PROGRAM FB_ApagadoCintas
VAR
END_VAR

IF POU_Contadores.iCintaProcesando = 0 THEN
	GVL_General.sBeltConveyor.bCintaAzul1 	:= FALSE;
	GVL_General.sBeltConveyor.bCintaVerde1	:= FALSE;
	GVL_General.sBeltConveyor.bCintaMetal1 	:= FALSE;
	GVL_General.sBeltConveyor.bCintaAzul2 	:= FALSE;
	GVL_General.sBeltConveyor.bCintaVerde2 	:= FALSE;
	GVL_General.sBeltConveyor.bCintaMetal2 	:= FALSE;
	GVL_General.sBeltConveyor.bSortingCintaDistribucion := FALSE;
END_IF

END_PROGRAM

(* stored: Version 1.1.0.1, ProductVersion 3.1.4024.12
   POU FB_ApagadoCintas: Id {405d3be8-2886-470d-a3cd-d9d8aa5b7439}, SpecialFunc None *)
